GVL_Objects.List_of_Recipes[3].Compress.Initial_Speed :=  ConfigData.Rec3_Compress_Initial_Speed;
GVL_Objects.List_of_Recipes[3].Compress.Initial_Distance := ConfigData.Rec3_Compress_Initial_Distance;
GVL_Objects.List_of_Recipes[3].Compress.Shield_Dwell := ConfigData.Rec3_Compress_Shield_Dwell;
GVL_Objects.List_of_Recipes[3].Compress.Relax_Distance := ConfigData.Rec3_Compress_Relax_Distance;
GVL_Objects.List_of_Recipes[3].Compress.Retract_Speed := ConfigData.Rec3_Compress_Retract_Speed;

GVL_Objects.List_of_Recipes[3].Pusher.Initial_Speed := ConfigData.Rec3_Pusher_Initial_Speed;
GVL_Objects.List_of_Recipes[3].Pusher.Initial_Distance := ConfigData.Rec3_Pusher_Initial_Distance;
GVL_Objects.List_of_Recipes[3].Pusher.Eject_Speed := ConfigData.Rec3_Pusher_Eject_Speed;
GVL_Objects.List_of_Recipes[3].Pusher.Eject_Distance := ConfigData.Rec3_Pusher_Eject_Distance;
GVL_Objects.List_of_Recipes[3].Pusher.Retract_Speed := ConfigData.Rec3_Pusher_Retract_Speed;

GVL_Objects.List_of_Recipes[3].Pusher.tamp_final_distance := ConfigData.Rec3_Pusher_tamp_final_distance;
GVL_Objects.List_of_Recipes[3].Pusher.tamp_final_speed := ConfigData.Rec3_Pusher_tamp_final_speed;
GVL_Objects.List_of_Recipes[3].Pusher.tamp_initial_distance := ConfigData.Rec3_Pusher_tamp_initial_distance;
GVL_Objects.List_of_Recipes[3].Pusher.tamp_initial_speed := ConfigData.Rec3_Pusher_tamp_initial_speed;

GVL_Objects.List_of_Recipes[3].Other.Compress_Home_Offset := ConfigData.Other3_Compress_Home_Offset;
GVL_Objects.List_of_Recipes[3].Other.Pusher_Home_Offset := ConfigData.Other3_Pusher_Home_Offset;
GVL_Objects.List_of_Recipes[3].Other.Shield_Home_Offset := ConfigData.Other3_Shield_Home_Offset;
GVL_Objects.List_of_Recipes[3].Other.Axis_Acceleration := ConfigData.Other3_Axis_Acceleration;
GVL_Objects.List_of_Recipes[3].Other.Axis_Deceleration := ConfigData.Other3_Axis_Deceleration;
GVL_Objects.List_of_Recipes[3].Other.Axis_Jerk := ConfigData.Other3_Axis_Jerk;
GVL_Objects.List_of_Recipes[3].Memory_Free := LREAL_TO_BOOL(ConfigData.Other3_Memory_Free);

GVL_Objects.List_of_Recipes[3].Clamp.Release_Instance := ConfigData.Clamp3_Release_Instance;

Rec4_Name_1:=ConfigData.Rec4_Name_1;								
Rec4_Name_2:=ConfigData.Rec4_Name_2;								
Rec4_Name_3:=ConfigData.Rec4_Name_3;								
Rec4_Name_4:=ConfigData.Rec4_Name_4;								
Rec4_Name_5:=ConfigData.Rec4_Name_5;
List_of_Recipes[4].Name := Recipe_mem_4;

GVL_Objects.List_of_Recipes[4].Shield.Retract_Speed := ConfigData.Rec4_Shield_Retract_Speed;
GVL_Objects.List_of_Recipes[4].Shield.Initial_Speed := ConfigData.Rec4_Shield_Initial_Speed;
GVL_Objects.List_of_Recipes[4].Shield.Initial_Distance := ConfigData.Rec4_Shield_Initial_Distance;

GVL_Objects.List_of_Recipes[4].Compress.Initial_Speed :=  ConfigData.Rec4_Compress_Initial_Speed;
GVL_Objects.List_of_Recipes[4].Compress.Initial_Distance := ConfigData.Rec4_Compress_Initial_Distance;
GVL_Objects.List_of_Recipes[4].Compress.Shield_Dwell := ConfigData.Rec4_Compress_Shield_Dwell;
GVL_Objects.List_of_Recipes[4].Compress.Relax_Distance := ConfigData.Rec4_Compress_Relax_Distance;
GVL_Objects.List_of_Recipes[4].Compress.Retract_Speed := ConfigData.Rec4_Compress_Retract_Speed;

GVL_Objects.List_of_Recipes[4].Pusher.Initial_Speed := ConfigData.Rec4_Pusher_Initial_Speed;
GVL_Objects.List_of_Recipes[4].Pusher.Initial_Distance := ConfigData.Rec4_Pusher_Initial_Distance;
GVL_Objects.List_of_Recipes[4].Pusher.Eject_Speed := ConfigData.Rec4_Pusher_Eject_Speed;
GVL_Objects.List_of_Recipes[4].Pusher.Eject_Distance := ConfigData.Rec4_Pusher_Eject_Distance;
GVL_Objects.List_of_Recipes[4].Pusher.Retract_Speed := ConfigData.Rec4_Pusher_Retract_Speed;

GVL_Objects.List_of_Recipes[4].Pusher.tamp_final_distance := ConfigData.Rec4_Pusher_tamp_final_distance;
GVL_Objects.List_of_Recipes[4].Pusher.tamp_final_speed := ConfigData.Rec4_Pusher_tamp_final_speed;
GVL_Objects.List_of_Recipes[4].Pusher.tamp_initial_distance := ConfigData.Rec4_Pusher_tamp_initial_distance;
GVL_Objects.List_of_Recipes[4].Pusher.tamp_initial_speed := ConfigData.Rec4_Pusher_tamp_initial_speed;

GVL_Objects.List_of_Recipes[4].Other.Compress_Home_Offset := ConfigData.Other4_Compress_Home_Offset;
GVL_Objects.List_of_Recipes[4].Other.Pusher_Home_Offset := ConfigData.Other4_Pusher_Home_Offset;
GVL_Objects.List_of_Recipes[4].Other.Shield_Home_Offset := ConfigData.Other4_Shield_Home_Offset;
GVL_Objects.List_of_Recipes[4].Other.Axis_Acceleration := ConfigData.Other4_Axis_Acceleration;
GVL_Objects.List_of_Recipes[4].Other.Axis_Deceleration := ConfigData.Other4_Axis_Deceleration;
GVL_Objects.List_of_Recipes[4].Other.Axis_Jerk := ConfigData.Other4_Axis_Jerk;
GVL_Objects.List_of_Recipes[4].Memory_Free := LREAL_TO_BOOL(ConfigData.Other4_Memory_Free);

GVL_Objects.List_of_Recipes[4].Clamp.Release_Instance := ConfigData.Clamp4_Release_Instance;

Rec5_Name_1:=ConfigData.Rec5_Name_1;								
Rec5_Name_2:=ConfigData.Rec5_Name_2;								
Rec5_Name_3:=ConfigData.Rec5_Name_3;								
Rec5_Name_4:=ConfigData.Rec5_Name_4;								
Rec5_Name_5:=ConfigData.Rec5_Name_5;
List_of_Recipes[5].Name := Recipe_mem_5;

GVL_Objects.List_of_Recipes[5].Shield.Retract_Speed := ConfigData.Rec5_Shield_Retract_Speed;
GVL_Objects.List_of_Recipes[5].Shield.Initial_Speed := ConfigData.Rec5_Shield_Initial_Speed;
GVL_Objects.List_of_Recipes[5].Shield.Initial_Distance := ConfigData.Rec5_Shield_Initial_Distance;

GVL_Objects.List_of_Recipes[5].Compress.Initial_Speed :=  ConfigData.Rec5_Compress_Initial_Speed;
GVL_Objects.List_of_Recipes[5].Compress.Initial_Distance := ConfigData.Rec5_Compress_Initial_Distance;
GVL_Objects.List_of_Recipes[5].Compress.Shield_Dwell := ConfigData.Rec5_Compress_Shield_Dwell;
GVL_Objects.List_of_Recipes[5].Compress.Relax_Distance := ConfigData.Rec5_Compress_Relax_Distance;
GVL_Objects.List_of_Recipes[5].Compress.Retract_Speed := ConfigData.Rec5_Compress_Retract_Speed;

GVL_Objects.List_of_Recipes[5].Pusher.Initial_Speed := ConfigData.Rec5_Pusher_Initial_Speed;
GVL_Objects.List_of_Recipes[5].Pusher.Initial_Distance := ConfigData.Rec5_Pusher_Initial_Distance;
GVL_Objects.List_of_Recipes[5].Pusher.Eject_Speed := ConfigData.Rec5_Pusher_Eject_Speed;
GVL_Objects.List_of_Recipes[5].Pusher.Eject_Distance := ConfigData.Rec5_Pusher_Eject_Distance;
GVL_Objects.List_of_Recipes[5].Pusher.Retract_Speed := ConfigData.Rec5_Pusher_Retract_Speed;

GVL_Objects.List_of_Recipes[5].Pusher.tamp_final_distance := ConfigData.Rec5_Pusher_tamp_final_distance;
GVL_Objects.List_of_Recipes[5].Pusher.tamp_final_speed := ConfigData.Rec5_Pusher_tamp_final_speed;
GVL_Objects.List_of_Recipes[5].Pusher.tamp_initial_distance := ConfigData.Rec5_Pusher_tamp_initial_distance;
GVL_Objects.List_of_Recipes[5].Pusher.tamp_initial_speed := ConfigData.Rec5_Pusher_tamp_initial_speed;

GVL_Objects.List_of_Recipes[5].Other.Compress_Home_Offset := ConfigData.Other5_Compress_Home_Offset;
GVL_Objects.List_of_Recipes[5].Other.Pusher_Home_Offset := ConfigData.Other5_Pusher_Home_Offset;
GVL_Objects.List_of_Recipes[5].Other.Shield_Home_Offset := ConfigData.Other5_Shield_Home_Offset;
GVL_Objects.List_of_Recipes[5].Other.Axis_Acceleration := ConfigData.Other5_Axis_Acceleration;
GVL_Objects.List_of_Recipes[5].Other.Axis_Deceleration := ConfigData.Other5_Axis_Deceleration;
GVL_Objects.List_of_Recipes[5].Other.Axis_Jerk := ConfigData.Other5_Axis_Jerk;
GVL_Objects.List_of_Recipes[5].Memory_Free := LREAL_TO_BOOL(ConfigData.Other5_Memory_Free);

GVL_Objects.List_of_Recipes[5].Clamp.Release_Instance := ConfigData.Clamp5_Release_Instance;

Rec6_Name_1:=ConfigData.Rec6_Name_1;								
Rec6_Name_2:=ConfigData.Rec6_Name_2;								
Rec6_Name_3:=ConfigData.Rec6_Name_3;								
Rec6_Name_4:=ConfigData.Rec6_Name_4;								
Rec6_Name_5:=ConfigData.Rec6_Name_5;
List_of_Recipes[6].Name := Recipe_mem_6;

GVL_Objects.List_of_Recipes[6].Shield.Retract_Speed := ConfigData.Rec6_Shield_Retract_Speed;
GVL_Objects.List_of_Recipes[6].Shield.Initial_Speed := ConfigData.Rec6_Shield_Initial_Speed;
GVL_Objects.List_of_Recipes[6].Shield.Initial_Distance := ConfigData.Rec6_Shield_Initial_Distance;

GVL_Objects.List_of_Recipes[6].Compress.Initial_Speed :=  ConfigData.Rec6_Compress_Initial_Speed;
GVL_Objects.List_of_Recipes[6].Compress.Initial_Distance := ConfigData.Rec6_Compress_Initial_Distance;
GVL_Objects.List_of_Recipes[6].Compress.Shield_Dwell := ConfigData.Rec6_Compress_Shield_Dwell;
GVL_Objects.List_of_Recipes[6].Compress.Relax_Distance := ConfigData.Rec6_Compress_Relax_Distance;
GVL_Objects.List_of_Recipes[6].Compress.Retract_Speed := ConfigData.Rec6_Compress_Retract_Speed;

GVL_Objects.List_of_Recipes[6].Pusher.Initial_Speed := ConfigData.Rec6_Pusher_Initial_Speed;
GVL_Objects.List_of_Recipes[6].Pusher.Initial_Distance := ConfigData.Rec6_Pusher_Initial_Distance;
GVL_Objects.List_of_Recipes[6].Pusher.Eject_Speed := ConfigData.Rec6_Pusher_Eject_Speed;
GVL_Objects.List_of_Recipes[6].Pusher.Eject_Distance := ConfigData.Rec6_Pusher_Eject_Distance;
GVL_Objects.List_of_Recipes[6].Pusher.Retract_Speed := ConfigData.Rec6_Pusher_Retract_Speed;

GVL_Objects.List_of_Recipes[6].Pusher.tamp_final_distance := ConfigData.Rec6_Pusher_tamp_final_distance;
GVL_Objects.List_of_Recipes[6].Pusher.tamp_final_speed := ConfigData.Rec6_Pusher_tamp_final_speed;
GVL_Objects.List_of_Recipes[6].Pusher.tamp_initial_distance := ConfigData.Rec6_Pusher_tamp_initial_distance;
GVL_Objects.List_of_Recipes[6].Pusher.tamp_initial_speed := ConfigData.Rec6_Pusher_tamp_initial_speed;

GVL_Objects.List_of_Recipes[6].Other.Compress_Home_Offset := ConfigData.Other6_Compress_Home_Offset;
GVL_Objects.List_of_Recipes[6].Other.Pusher_Home_Offset := ConfigData.Other6_Pusher_Home_Offset;
GVL_Objects.List_of_Recipes[6].Other.Shield_Home_Offset := ConfigData.Other6_Shield_Home_Offset;
GVL_Objects.List_of_Recipes[6].Other.Axis_Acceleration := ConfigData.Other6_Axis_Acceleration;
GVL_Objects.List_of_Recipes[6].Other.Axis_Deceleration := ConfigData.Other6_Axis_Deceleration;
GVL_Objects.List_of_Recipes[6].Other.Axis_Jerk := ConfigData.Other6_Axis_Jerk;
GVL_Objects.List_of_Recipes[6].Memory_Free := LREAL_TO_BOOL(ConfigData.Other6_Memory_Free);

GVL_Objects.List_of_Recipes[6].Clamp.Release_Instance := ConfigData.Clamp6_Release_Instance;

Rec7_Name_1:=ConfigData.Rec7_Name_1;								
Rec7_Name_2:=ConfigData.Rec7_Name_2;								
Rec7_Name_3:=ConfigData.Rec7_Name_3;								
Rec7_Name_4:=ConfigData.Rec7_Name_4;								
Rec7_Name_5:=ConfigData.Rec7_Name_5;
List_of_Recipes[7].Name := Recipe_mem_7;

GVL_Objects.List_of_Recipes[7].Shield.Retract_Speed := ConfigData.Rec7_Shield_Retract_Speed;
GVL_Objects.List_of_Recipes[7].Shield.Initial_Speed := ConfigData.Rec7_Shield_Initial_Speed;
GVL_Objects.List_of_Recipes[7].Shield.Initial_Distance := ConfigData.Rec7_Shield_Initial_Distance;

GVL_Objects.List_of_Recipes[7].Compress.Initial_Speed :=  ConfigData.Rec7_Compress_Initial_Speed;
GVL_Objects.List_of_Recipes[7].Compress.Initial_Distance := ConfigData.Rec7_Compress_Initial_Distance;
GVL_Objects.List_of_Recipes[7].Compress.Shield_Dwell := ConfigData.Rec7_Compress_Shield_Dwell;
GVL_Objects.List_of_Recipes[7].Compress.Relax_Distance := ConfigData.Rec7_Compress_Relax_Distance;
GVL_Objects.List_of_Recipes[7].Compress.Retract_Speed := ConfigData.Rec7_Compress_Retract_Speed;

GVL_Objects.List_of_Recipes[7].Pusher.Initial_Speed := ConfigData.Rec7_Pusher_Initial_Speed;
GVL_Objects.List_of_Recipes[7].Pusher.Initial_Distance := ConfigData.Rec7_Pusher_Initial_Distance;
GVL_Objects.List_of_Recipes[7].Pusher.Eject_Speed := ConfigData.Rec7_Pusher_Eject_Speed;
GVL_Objects.List_of_Recipes[7].Pusher.Eject_Distance := ConfigData.Rec7_Pusher_Eject_Distance;
GVL_Objects.List_of_Recipes[7].Pusher.Retract_Speed := ConfigData.Rec7_Pusher_Retract_Speed;

GVL_Objects.List_of_Recipes[7].Pusher.tamp_final_distance := ConfigData.Rec7_Pusher_tamp_final_distance;
GVL_Objects.List_of_Recipes[7].Pusher.tamp_final_speed := ConfigData.Rec7_Pusher_tamp_final_speed;
GVL_Objects.List_of_Recipes[7].Pusher.tamp_initial_distance := ConfigData.Rec7_Pusher_tamp_initial_distance;
GVL_Objects.List_of_Recipes[7].Pusher.tamp_initial_speed := ConfigData.Rec7_Pusher_tamp_initial_speed;

GVL_Objects.List_of_Recipes[7].Other.Compress_Home_Offset := ConfigData.Other7_Compress_Home_Offset;
GVL_Objects.List_of_Recipes[7].Other.Pusher_Home_Offset := ConfigData.Other7_Pusher_Home_Offset;
GVL_Objects.List_of_Recipes[7].Other.Shield_Home_Offset := ConfigData.Other7_Shield_Home_Offset;
GVL_Objects.List_of_Recipes[7].Other.Axis_Acceleration := ConfigData.Other7_Axis_Acceleration;
GVL_Objects.List_of_Recipes[7].Other.Axis_Deceleration := ConfigData.Other7_Axis_Deceleration;
GVL_Objects.List_of_Recipes[7].Other.Axis_Jerk := ConfigData.Other7_Axis_Jerk;
GVL_Objects.List_of_Recipes[7].Memory_Free := LREAL_TO_BOOL(ConfigData.Other7_Memory_Free);

GVL_Objects.List_of_Recipes[7].Clamp.Release_Instance := ConfigData.Clamp7_Release_Instance;

Rec8_Name_1:=ConfigData.Rec8_Name_1;								
Rec8_Name_2:=ConfigData.Rec8_Name_2;								
Rec8_Name_3:=ConfigData.Rec8_Name_3;								
Rec8_Name_4:=ConfigData.Rec8_Name_4;								
Rec8_Name_5:=ConfigData.Rec8_Name_5;
List_of_Recipes[8].Name := Recipe_mem_8;

GVL_Objects.List_of_Recipes[8].Shield.Retract_Speed := ConfigData.Rec8_Shield_Retract_Speed;
GVL_Objects.List_of_Recipes[8].Shield.Initial_Speed := ConfigData.Rec8_Shield_Initial_Speed;
GVL_Objects.List_of_Recipes[8].Shield.Initial_Distance := ConfigData.Rec8_Shield_Initial_Distance;

GVL_Objects.List_of_Recipes[8].Compress.Initial_Speed :=  ConfigData.Rec8_Compress_Initial_Speed;
GVL_Objects.List_of_Recipes[8].Compress.Initial_Distance := ConfigData.Rec8_Compress_Initial_Distance;
GVL_Objects.List_of_Recipes[8].Compress.Shield_Dwell := ConfigData.Rec8_Compress_Shield_Dwell;
GVL_Objects.List_of_Recipes[8].Compress.Relax_Distance := ConfigData.Rec8_Compress_Relax_Distance;
GVL_Objects.List_of_Recipes[8].Compress.Retract_Speed := ConfigData.Rec8_Compress_Retract_Speed;

GVL_Objects.List_of_Recipes[8].Pusher.Initial_Speed := ConfigData.Rec8_Pusher_Initial_Speed;
GVL_Objects.List_of_Recipes[8].Pusher.Initial_Distance := ConfigData.Rec8_Pusher_Initial_Distance;
GVL_Objects.List_of_Recipes[8].Pusher.Eject_Speed := ConfigData.Rec8_Pusher_Eject_Speed;
GVL_Objects.List_of_Recipes[8].Pusher.Eject_Distance := ConfigData.Rec8_Pusher_Eject_Distance;
GVL_Objects.List_of_Recipes[8].Pusher.Retract_Speed := ConfigData.Rec8_Pusher_Retract_Speed;

GVL_Objects.List_of_Recipes[8].Pusher.tamp_final_distance := ConfigData.Rec8_Pusher_tamp_final_distance;
GVL_Objects.List_of_Recipes[8].Pusher.tamp_final_speed := ConfigData.Rec8_Pusher_tamp_final_speed;
GVL_Objects.List_of_Recipes[8].Pusher.tamp_initial_distance := ConfigData.Rec8_Pusher_tamp_initial_distance;
GVL_Objects.List_of_Recipes[8].Pusher.tamp_initial_speed := ConfigData.Rec8_Pusher_tamp_initial_speed;

GVL_Objects.List_of_Recipes[8].Other.Compress_Home_Offset := ConfigData.Other8_Compress_Home_Offset;
GVL_Objects.List_of_Recipes[8].Other.Pusher_Home_Offset := ConfigData.Other8_Pusher_Home_Offset;
GVL_Objects.List_of_Recipes[8].Other.Shield_Home_Offset := ConfigData.Other8_Shield_Home_Offset;
GVL_Objects.List_of_Recipes[8].Other.Axis_Acceleration := ConfigData.Other8_Axis_Acceleration;
GVL_Objects.List_of_Recipes[8].Other.Axis_Deceleration := ConfigData.Other8_Axis_Deceleration;
GVL_Objects.List_of_Recipes[8].Other.Axis_Jerk := ConfigData.Other8_Axis_Jerk;
GVL_Objects.List_of_Recipes[8].Memory_Free := LREAL_TO_BOOL(ConfigData.Other8_Memory_Free);

GVL_Objects.List_of_Recipes[8].Clamp.Release_Instance := ConfigData.Clamp8_Release_Instance;

Rec9_Name_1:=ConfigData.Rec9_Name_1;								
Rec9_Name_2:=ConfigData.Rec9_Name_2;								
Rec9_Name_3:=ConfigData.Rec9_Name_3;								
Rec9_Name_4:=ConfigData.Rec9_Name_4;								
Rec9_Name_5:=ConfigData.Rec9_Name_5;
List_of_Recipes[9].Name := Recipe_mem_9;

GVL_Objects.List_of_Recipes[9].Shield.Retract_Speed := ConfigData.Rec9_Shield_Retract_Speed;
GVL_Objects.List_of_Recipes[9].Shield.Initial_Speed := ConfigData.Rec9_Shield_Initial_Speed;
GVL_Objects.List_of_Recipes[9].Shield.Initial_Distance := ConfigData.Rec9_Shield_Initial_Distance;

GVL_Objects.List_of_Recipes[9].Compress.Initial_Speed :=  ConfigData.Rec9_Compress_Initial_Speed;
GVL_Objects.List_of_Recipes[9].Compress.Initial_Distance := ConfigData.Rec9_Compress_Initial_Distance;
GVL_Objects.List_of_Recipes[9].Compress.Shield_Dwell := ConfigData.Rec9_Compress_Shield_Dwell;
GVL_Objects.List_of_Recipes[9].Compress.Relax_Distance := ConfigData.Rec9_Compress_Relax_Distance;
GVL_Objects.List_of_Recipes[9].Compress.Retract_Speed := ConfigData.Rec9_Compress_Retract_Speed;

GVL_Objects.List_of_Recipes[9].Pusher.Initial_Speed := ConfigData.Rec9_Pusher_Initial_Speed;
GVL_Objects.List_of_Recipes[9].Pusher.Initial_Distance := ConfigData.Rec9_Pusher_Initial_Distance;
GVL_Objects.List_of_Recipes[9].Pusher.Eject_Speed := ConfigData.Rec9_Pusher_Eject_Speed;
GVL_Objects.List_of_Recipes[9].Pusher.Eject_Distance := ConfigData.Rec9_Pusher_Eject_Distance;
GVL_Objects.List_of_Recipes[9].Pusher.Retract_Speed := ConfigData.Rec9_Pusher_Retract_Speed;

GVL_Objects.List_of_Recipes[9].Pusher.tamp_final_distance := ConfigData.Rec9_Pusher_tamp_final_distance;
GVL_Objects.List_of_Recipes[9].Pusher.tamp_final_speed := ConfigData.Rec9_Pusher_tamp_final_speed;
GVL_Objects.List_of_Recipes[9].Pusher.tamp_initial_distance := ConfigData.Rec9_Pusher_tamp_initial_distance;
GVL_Objects.List_of_Recipes[9].Pusher.tamp_initial_speed := ConfigData.Rec9_Pusher_tamp_initial_speed;

GVL_Objects.List_of_Recipes[9].Other.Compress_Home_Offset := ConfigData.Other9_Compress_Home_Offset;
GVL_Objects.List_of_Recipes[9].Other.Pusher_Home_Offset := ConfigData.Other9_Pusher_Home_Offset;
GVL_Objects.List_of_Recipes[9].Other.Shield_Home_Offset := ConfigData.Other9_Shield_Home_Offset;
GVL_Objects.List_of_Recipes[9].Other.Axis_Acceleration := ConfigData.Other9_Axis_Acceleration;
GVL_Objects.List_of_Recipes[9].Other.Axis_Deceleration := ConfigData.Other9_Axis_Deceleration;
GVL_Objects.List_of_Recipes[9].Other.Axis_Jerk := ConfigData.Other9_Axis_Jerk;
GVL_Objects.List_of_Recipes[9].Memory_Free := LREAL_TO_BOOL(ConfigData.Other9_Memory_Free);

GVL_Objects.List_of_Recipes[9].Clamp.Release_Instance := ConfigData.Clamp9_Release_Instance;

Rec10_Name_1:=ConfigData.Rec10_Name_1;								
Rec10_Name_2:=ConfigData.Rec10_Name_2;								
Rec10_Name_3:=ConfigData.Rec10_Name_3;								
Rec10_Name_4:=ConfigData.Rec10_Name_4;								
Rec10_Name_5:=ConfigData.Rec10_Name_5;
List_of_Recipes[10].Name := Recipe_mem_10;

GVL_Objects.List_of_Recipes[10].Shield.Retract_Speed := ConfigData.Rec10_Shield_Retract_Speed;
GVL_Objects.List_of_Recipes[10].Shield.Initial_Speed := ConfigData.Rec10_Shield_Initial_Speed;
GVL_Objects.List_of_Recipes[10].Shield.Initial_Distance := ConfigData.Rec10_Shield_Initial_Distance;

GVL_Objects.List_of_Recipes[10].Compress.Initial_Speed :=  ConfigData.Rec10_Compress_Initial_Speed;
GVL_Objects.List_of_Recipes[10].Compress.Initial_Distance := ConfigData.Rec10_Compress_Initial_Distance;
GVL_Objects.List_of_Recipes[10].Compress.Shield_Dwell := ConfigData.Rec10_Compress_Shield_Dwell;
GVL_Objects.List_of_Recipes[10].Compress.Relax_Distance := ConfigData.Rec10_Compress_Relax_Distance;
GVL_Objects.List_of_Recipes[10].Compress.Retract_Speed := ConfigData.Rec10_Compress_Retract_Speed;

GVL_Objects.List_of_Recipes[10].Pusher.Initial_Speed := ConfigData.Rec10_Pusher_Initial_Speed;
GVL_Objects.List_of_Recipes[10].Pusher.Initial_Distance := ConfigData.Rec10_Pusher_Initial_Distance;
GVL_Objects.List_of_Recipes[10].Pusher.Eject_Speed := ConfigData.Rec10_Pusher_Eject_Speed;
GVL_Objects.List_of_Recipes[10].Pusher.Eject_Distance := ConfigData.Rec10_Pusher_Eject_Distance;
GVL_Objects.List_of_Recipes[10].Pusher.Retract_Speed := ConfigData.Rec10_Pusher_Retract_Speed;

GVL_Objects.List_of_Recipes[10].Pusher.tamp_final_distance := ConfigData.Rec10_Pusher_tamp_final_distance;
GVL_Objects.List_of_Recipes[10].Pusher.tamp_final_speed := ConfigData.Rec10_Pusher_tamp_final_speed;
GVL_Objects.List_of_Recipes[10].Pusher.tamp_initial_distance := ConfigData.Rec10_Pusher_tamp_initial_distance;
GVL_Objects.List_of_Recipes[10].Pusher.tamp_initial_speed := ConfigData.Rec10_Pusher_tamp_initial_speed;

GVL_Objects.List_of_Recipes[10].Other.Compress_Home_Offset := ConfigData.Other10_Compress_Home_Offset;
GVL_Objects.List_of_Recipes[10].Other.Pusher_Home_Offset := ConfigData.Other10_Pusher_Home_Offset;
GVL_Objects.List_of_Recipes[10].Other.Shield_Home_Offset := ConfigData.Other10_Shield_Home_Offset;
GVL_Objects.List_of_Recipes[10].Other.Axis_Acceleration := ConfigData.Other10_Axis_Acceleration;
GVL_Objects.List_of_Recipes[10].Other.Axis_Deceleration := ConfigData.Other10_Axis_Deceleration;
GVL_Objects.List_of_Recipes[10].Other.Axis_Jerk := ConfigData.Other10_Axis_Jerk;
GVL_Objects.List_of_Recipes[10].Memory_Free := LREAL_TO_BOOL(ConfigData.Other10_Memory_Free);

GVL_Objects.List_of_Recipes[10].Clamp.Release_Instance := ConfigData.Clamp10_Release_Instance;


//limits
GVL_Zenon.limits_save.max_limit_Compress := ConfigData.con_max_limit_Compress ; 					
GVL_Zenon.limits_save.max_limit_Shield := ConfigData.con_max_limit_Shield; 					
GVL_Zenon.limits_save.max_limit_Pusher := ConfigData.con_max_limit_Pusher;					
GVL_Zenon.limits_save.max_pusher_shield_diff := ConfigData.con_max_pusher_shield_diff;
END_METHOD

METHOD CopyConfigSettingsToGlobal : BOOL
VAR_INPUT
END_VAR
END_METHOD

METHOD CopyGlobalRecipiesToConfig : BOOL
VAR_INPUT
END_VAR
//ConfigData.Rec1_Name := GVL_Objects.List_of_Recipes[1].Name;

 
Recipe_mem_1:= List_of_Recipes[1].Name;

ConfigData.Rec1_Name_1:=Rec1_Name_1;								
ConfigData.Rec1_Name_2:=Rec1_Name_2;								
ConfigData.Rec1_Name_3:=Rec1_Name_3;								
ConfigData.Rec1_Name_4:=Rec1_Name_4;								
ConfigData.Rec1_Name_5:=Rec1_Name_5;	

ConfigData.Rec1_Shield_Retract_Speed := GVL_Objects.List_of_Recipes[1].Shield.Retract_Speed;
ConfigData.Rec1_Shield_Initial_Speed := GVL_Objects.List_of_Recipes[1].Shield.Initial_Speed;
ConfigData.Rec1_Shield_Initial_Distance := GVL_Objects.List_of_Recipes[1].Shield.Initial_distance;

ConfigData.Rec1_Compress_Initial_Speed := GVL_Objects.List_of_Recipes[1].Compress.Initial_Speed;
ConfigData.Rec1_Compress_Initial_Distance := GVL_Objects.List_of_Recipes[1].Compress.Initial_Distance;
ConfigData.Rec1_Compress_Shield_Dwell := GVL_Objects.List_of_Recipes[1].Compress.Shield_Dwell;
ConfigData.Rec1_Compress_Relax_Distance := GVL_Objects.List_of_Recipes[1].Compress.Relax_Distance;
ConfigData.Rec1_Compress_Retract_Speed := GVL_Objects.List_of_Recipes[1].Compress.Retract_Speed;


ConfigData.Rec1_Pusher_Initial_Speed := GVL_Objects.List_of_Recipes[1].Pusher.Initial_Speed;
ConfigData.Rec1_Pusher_Initial_Distance := GVL_Objects.List_of_Recipes[1].Pusher.Initial_Distance;
ConfigData.Rec1_Pusher_Eject_Speed := GVL_Objects.List_of_Recipes[1].Pusher.Eject_Speed;
ConfigData.Rec1_Pusher_Eject_Distance := GVL_Objects.List_of_Recipes[1].Pusher.Eject_Distance;
ConfigData.Rec1_Pusher_Retract_Speed := GVL_Objects.List_of_Recipes[1].Pusher.Retract_Speed;

ConfigData.Rec1_Pusher_tamp_initial_distance := GVL_Objects.List_of_Recipes[1].Pusher.tamp_initial_distance;
ConfigData.Rec1_Pusher_tamp_initial_speed := GVL_Objects.List_of_Recipes[1].Pusher.tamp_initial_speed;
ConfigData.Rec1_Pusher_tamp_final_distance := GVL_Objects.List_of_Recipes[1].Pusher.tamp_final_distance;
ConfigData.Rec1_Pusher_tamp_final_speed := GVL_Objects.List_of_Recipes[1].Pusher.tamp_final_speed;

ConfigData.Other1_Compress_Home_Offset := GVL_Objects.List_of_Recipes[1].Other.Compress_Home_Offset;
ConfigData.Other1_Pusher_Home_Offset := GVL_Objects.List_of_Recipes[1].Other.Pusher_Home_Offset;
ConfigData.Other1_Shield_Home_Offset := GVL_Objects.List_of_Recipes[1].Other.Shield_Home_Offset;
ConfigData.Other1_Axis_Acceleration := GVL_Objects.List_of_Recipes[1].Other.Axis_Acceleration;
ConfigData.Other1_Axis_Deceleration :=GVL_Objects.List_of_Recipes[1].Other.Axis_Deceleration;
ConfigData.Other1_Axis_Jerk := GVL_Objects.List_of_Recipes[1].Other.Axis_Jerk;
ConfigData.Other1_Memory_Free := BOOL_TO_LREAL(GVL_Objects.List_of_Recipes[1].Memory_Free);

ConfigData.Clamp1_Release_Instance := GVL_Objects.List_of_Recipes[1].Clamp.Release_Instance;

Recipe_mem_2:= List_of_Recipes[2].Name;
ConfigData.Rec2_Name_1:=Rec2_Name_1;								
ConfigData.Rec2_Name_2:=Rec2_Name_2;								
ConfigData.Rec2_Name_3:=Rec2_Name_3;								
ConfigData.Rec2_Name_4:=Rec2_Name_4;								
ConfigData.Rec2_Name_5:=Rec2_Name_5;

ConfigData.Rec2_Shield_Retract_Speed := GVL_Objects.List_of_Recipes[2].Shield.Retract_Speed;
ConfigData.Rec2_Shield_Initial_Speed := GVL_Objects.List_of_Recipes[2].Shield.Initial_Speed;
ConfigData.Rec2_Shield_Initial_Distance := GVL_Objects.List_of_Recipes[2].Shield.Initial_distance;

ConfigData.Rec2_Compress_Initial_Speed := GVL_Objects.List_of_Recipes[2].Compress.Initial_Speed;
ConfigData.Rec2_Compress_Initial_Distance := GVL_Objects.List_of_Recipes[2].Compress.Initial_Distance;
ConfigData.Rec2_Compress_Shield_Dwell := GVL_Objects.List_of_Recipes[2].Compress.Shield_Dwell;
ConfigData.Rec2_Compress_Relax_Distance := GVL_Objects.List_of_Recipes[2].Compress.Relax_Distance;
ConfigData.Rec2_Compress_Retract_Speed := GVL_Objects.List_of_Recipes[2].Compress.Retract_Speed;

ConfigData.Rec2_Pusher_Initial_Speed := GVL_Objects.List_of_Recipes[2].Pusher.Initial_Speed;
ConfigData.Rec2_Pusher_Initial_Distance := GVL_Objects.List_of_Recipes[2].Pusher.Initial_Distance;
ConfigData.Rec2_Pusher_Eject_Speed := GVL_Objects.List_of_Recipes[2].Pusher.Eject_Speed;
ConfigData.Rec2_Pusher_Eject_Distance := GVL_Objects.List_of_Recipes[2].Pusher.Eject_Distance;
ConfigData.Rec2_Pusher_Retract_Speed := GVL_Objects.List_of_Recipes[2].Pusher.Retract_Speed;

ConfigData.Rec2_Pusher_tamp_initial_distance := GVL_Objects.List_of_Recipes[2].Pusher.tamp_initial_distance;
ConfigData.Rec2_Pusher_tamp_initial_speed := GVL_Objects.List_of_Recipes[2].Pusher.tamp_initial_speed;
ConfigData.Rec2_Pusher_tamp_final_distance := GVL_Objects.List_of_Recipes[2].Pusher.tamp_final_distance;
ConfigData.Rec2_Pusher_tamp_final_speed := GVL_Objects.List_of_Recipes[2].Pusher.tamp_final_speed;

ConfigData.Other2_Compress_Home_Offset := GVL_Objects.List_of_Recipes[2].Other.Compress_Home_Offset;
ConfigData.Other2_Pusher_Home_Offset := GVL_Objects.List_of_Recipes[2].Other.Pusher_Home_Offset;
ConfigData.Other2_Shield_Home_Offset := GVL_Objects.List_of_Recipes[2].Other.Shield_Home_Offset;
ConfigData.Other2_Axis_Acceleration := GVL_Objects.List_of_Recipes[2].Other.Axis_Acceleration;
ConfigData.Other2_Axis_Deceleration :=GVL_Objects.List_of_Recipes[2].Other.Axis_Deceleration;
ConfigData.Other2_Axis_Jerk := GVL_Objects.List_of_Recipes[2].Other.Axis_Jerk;
ConfigData.Other2_Memory_Free := BOOL_TO_LREAL(GVL_Objects.List_of_Recipes[2].Memory_Free);

ConfigData.Clamp2_Release_Instance := GVL_Objects.List_of_Recipes[2].Clamp.Release_Instance;

Recipe_mem_3:= List_of_Recipes[3].Name;
ConfigData.Rec3_Name_1:=Rec3_Name_1;								
ConfigData.Rec3_Name_2:=Rec3_Name_2;								
ConfigData.Rec3_Name_3:=Rec3_Name_3;								
ConfigData.Rec3_Name_4:=Rec3_Name_4;								
ConfigData.Rec3_Name_5:=Rec3_Name_5;

ConfigData.Rec3_Shield_Retract_Speed := GVL_Objects.List_of_Recipes[3].Shield.Retract_Speed;
ConfigData.Rec3_Shield_Initial_Speed := GVL_Objects.List_of_Recipes[3].Shield.Initial_Speed;
ConfigData.Rec3_Shield_Initial_Distance := GVL_Objects.List_of_Recipes[3].Shield.Initial_distance;

ConfigData.Rec3_Compress_Initial_Speed := GVL_Objects.List_of_Recipes[3].Compress.Initial_Speed;
ConfigData.Rec3_Compress_Initial_Distance := GVL_Objects.List_of_Recipes[3].Compress.Initial_Distance;
ConfigData.Rec3_Compress_Shield_Dwell := GVL_Objects.List_of_Recipes[3].Compress.Shield_Dwell;
ConfigData.Rec3_Compress_Relax_Distance := GVL_Objects.List_of_Recipes[3].Compress.Relax_Distance;
ConfigData.Rec3_Compress_Retract_Speed := GVL_Objects.List_of_Recipes[3].Compress.Retract_Speed;

ConfigData.Rec3_Pusher_Initial_Speed := GVL_Objects.List_of_Recipes[3].Pusher.Initial_Speed;
ConfigData.Rec3_Pusher_Initial_Distance := GVL_Objects.List_of_Recipes[3].Pusher.Initial_Distance;
ConfigData.Rec3_Pusher_Eject_Speed := GVL_Objects.List_of_Recipes[3].Pusher.Eject_Speed;
ConfigData.Rec3_Pusher_Eject_Distance := GVL_Objects.List_of_Recipes[3].Pusher.Eject_Distance;
ConfigData.Rec3_Pusher_Retract_Speed := GVL_Objects.List_of_Recipes[3].Pusher.Retract_Speed;

ConfigData.Rec3_Pusher_tamp_initial_distance := GVL_Objects.List_of_Recipes[3].Pusher.tamp_initial_distance;
ConfigData.Rec3_Pusher_tamp_initial_speed := GVL_Objects.List_of_Recipes[3].Pusher.tamp_initial_speed;
ConfigData.Rec3_Pusher_tamp_final_distance := GVL_Objects.List_of_Recipes[3].Pusher.tamp_final_distance;
ConfigData.Rec3_Pusher_tamp_final_speed := GVL_Objects.List_of_Recipes[3].Pusher.tamp_final_speed;

ConfigData.Other3_Compress_Home_Offset := GVL_Objects.List_of_Recipes[3].Other.Compress_Home_Offset;
ConfigData.Other3_Pusher_Home_Offset := GVL_Objects.List_of_Recipes[3].Other.Pusher_Home_Offset;
ConfigData.Other3_Shield_Home_Offset := GVL_Objects.List_of_Recipes[3].Other.Shield_Home_Offset;
ConfigData.Other3_Axis_Acceleration := GVL_Objects.List_of_Recipes[3].Other.Axis_Acceleration;
ConfigData.Other3_Axis_Deceleration :=GVL_Objects.List_of_Recipes[3].Other.Axis_Deceleration;
ConfigData.Other3_Axis_Jerk := GVL_Objects.List_of_Recipes[3].Other.Axis_Jerk;
ConfigData.Other3_Memory_Free := BOOL_TO_LREAL(GVL_Objects.List_of_Recipes[3].Memory_Free);

ConfigData.Clamp3_Release_Instance := GVL_Objects.List_of_Recipes[3].Clamp.Release_Instance;

Recipe_mem_4:= List_of_Recipes[4].Name;
ConfigData.Rec4_Name_1:=Rec4_Name_1;								
ConfigData.Rec4_Name_2:=Rec4_Name_2;								
ConfigData.Rec4_Name_3:=Rec4_Name_3;								
ConfigData.Rec4_Name_4:=Rec4_Name_4;								
ConfigData.Rec4_Name_5:=Rec4_Name_5;

ConfigData.Rec4_Shield_Retract_Speed := GVL_Objects.List_of_Recipes[4].Shield.Retract_Speed;
ConfigData.Rec4_Shield_Initial_Speed := GVL_Objects.List_of_Recipes[4].Shield.Initial_Speed;
ConfigData.Rec4_Shield_Initial_Distance := GVL_Objects.List_of_Recipes[4].Shield.Initial_distance;

ConfigData.Rec4_Compress_Initial_Speed := GVL_Objects.List_of_Recipes[4].Compress.Initial_Speed;
ConfigData.Rec4_Compress_Initial_Distance := GVL_Objects.List_of_Recipes[4].Compress.Initial_Distance;
ConfigData.Rec4_Compress_Shield_Dwell := GVL_Objects.List_of_Recipes[4].Compress.Shield_Dwell;
ConfigData.Rec4_Compress_Relax_Distance := GVL_Objects.List_of_Recipes[4].Compress.Relax_Distance;
ConfigData.Rec4_Compress_Retract_Speed := GVL_Objects.List_of_Recipes[4].Compress.Retract_Speed;

ConfigData.Rec4_Pusher_Initial_Speed := GVL_Objects.List_of_Recipes[4].Pusher.Initial_Speed;
ConfigData.Rec4_Pusher_Initial_Distance := GVL_Objects.List_of_Recipes[4].Pusher.Initial_Distance;
ConfigData.Rec4_Pusher_Eject_Speed := GVL_Objects.List_of_Recipes[4].Pusher.Eject_Speed;
ConfigData.Rec4_Pusher_Eject_Distance := GVL_Objects.List_of_Recipes[4].Pusher.Eject_Distance;
ConfigData.Rec4_Pusher_Retract_Speed := GVL_Objects.List_of_Recipes[4].Pusher.Retract_Speed;

ConfigData.Rec4_Pusher_tamp_initial_distance := GVL_Objects.List_of_Recipes[4].Pusher.tamp_initial_distance;
ConfigData.Rec4_Pusher_tamp_initial_speed := GVL_Objects.List_of_Recipes[4].Pusher.tamp_initial_speed;
ConfigData.Rec4_Pusher_tamp_final_distance := GVL_Objects.List_of_Recipes[4].Pusher.tamp_final_distance;
ConfigData.Rec4_Pusher_tamp_final_speed := GVL_Objects.List_of_Recipes[4].Pusher.tamp_final_speed;

ConfigData.Other4_Compress_Home_Offset := GVL_Objects.List_of_Recipes[4].Other.Compress_Home_Offset;
ConfigData.Other4_Pusher_Home_Offset := GVL_Objects.List_of_Recipes[4].Other.Pusher_Home_Offset;
ConfigData.Other4_Shield_Home_Offset := GVL_Objects.List_of_Recipes[4].Other.Shield_Home_Offset;
ConfigData.Other4_Axis_Acceleration := GVL_Objects.List_of_Recipes[4].Other.Axis_Acceleration;
ConfigData.Other4_Axis_Deceleration :=GVL_Objects.List_of_Recipes[4].Other.Axis_Deceleration;
ConfigData.Other4_Axis_Jerk := GVL_Objects.List_of_Recipes[4].Other.Axis_Jerk;
ConfigData.Other4_Memory_Free := BOOL_TO_LREAL(GVL_Objects.List_of_Recipes[4].Memory_Free);

ConfigData.Clamp4_Release_Instance := GVL_Objects.List_of_Recipes[4].Clamp.Release_Instance;

Recipe_mem_5:= List_of_Recipes[5].Name;
ConfigData.Rec5_Name_1:=Rec5_Name_1;								
ConfigData.Rec5_Name_2:=Rec5_Name_2;								
ConfigData.Rec5_Name_3:=Rec5_Name_3;								
ConfigData.Rec5_Name_4:=Rec5_Name_4;								
ConfigData.Rec5_Name_5:=Rec5_Name_5;

ConfigData.Rec5_Shield_Retract_Speed := GVL_Objects.List_of_Recipes[5].Shield.Retract_Speed;
ConfigData.Rec5_Shield_Initial_Speed := GVL_Objects.List_of_Recipes[5].Shield.Initial_Speed;
ConfigData.Rec5_Shield_Initial_Distance := GVL_Objects.List_of_Recipes[5].Shield.Initial_distance;

ConfigData.Rec5_Compress_Initial_Speed := GVL_Objects.List_of_Recipes[5].Compress.Initial_Speed;
ConfigData.Rec5_Compress_Initial_Distance := GVL_Objects.List_of_Recipes[5].Compress.Initial_Distance;
ConfigData.Rec5_Compress_Shield_Dwell := GVL_Objects.List_of_Recipes[5].Compress.Shield_Dwell;
ConfigData.Rec5_Compress_Relax_Distance := GVL_Objects.List_of_Recipes[5].Compress.Relax_Distance;
ConfigData.Rec5_Compress_Retract_Speed := GVL_Objects.List_of_Recipes[5].Compress.Retract_Speed;

ConfigData.Rec5_Pusher_Initial_Speed := GVL_Objects.List_of_Recipes[5].Pusher.Initial_Speed;
ConfigData.Rec5_Pusher_Initial_Distance := GVL_Objects.List_of_Recipes[5].Pusher.Initial_Distance;
ConfigData.Rec5_Pusher_Eject_Speed := GVL_Objects.List_of_Recipes[5].Pusher.Eject_Speed;
ConfigData.Rec5_Pusher_Eject_Distance := GVL_Objects.List_of_Recipes[5].Pusher.Eject_Distance;
ConfigData.Rec5_Pusher_Retract_Speed := GVL_Objects.List_of_Recipes[5].Pusher.Retract_Speed;

ConfigData.Rec5_Pusher_tamp_initial_distance := GVL_Objects.List_of_Recipes[5].Pusher.tamp_initial_distance;
ConfigData.Rec5_Pusher_tamp_initial_speed := GVL_Objects.List_of_Recipes[5].Pusher.tamp_initial_speed;
ConfigData.Rec5_Pusher_tamp_final_distance := GVL_Objects.List_of_Recipes[5].Pusher.tamp_final_distance;
ConfigData.Rec5_Pusher_tamp_final_speed := GVL_Objects.List_of_Recipes[5].Pusher.tamp_final_speed;

ConfigData.Other5_Compress_Home_Offset := GVL_Objects.List_of_Recipes[5].Other.Compress_Home_Offset;
ConfigData.Other5_Pusher_Home_Offset := GVL_Objects.List_of_Recipes[5].Other.Pusher_Home_Offset;
ConfigData.Other5_Shield_Home_Offset := GVL_Objects.List_of_Recipes[5].Other.Shield_Home_Offset;
ConfigData.Other5_Axis_Acceleration := GVL_Objects.List_of_Recipes[5].Other.Axis_Acceleration;
ConfigData.Other5_Axis_Deceleration :=GVL_Objects.List_of_Recipes[5].Other.Axis_Deceleration;
ConfigData.Other5_Axis_Jerk := GVL_Objects.List_of_Recipes[5].Other.Axis_Jerk;
ConfigData.Other5_Memory_Free := BOOL_TO_LREAL(GVL_Objects.List_of_Recipes[5].Memory_Free);

ConfigData.Clamp5_Release_Instance := GVL_Objects.List_of_Recipes[5].Clamp.Release_Instance;

Recipe_mem_6:= List_of_Recipes[6].Name;
ConfigData.Rec6_Name_1:=Rec6_Name_1;								
ConfigData.Rec6_Name_2:=Rec6_Name_2;								
ConfigData.Rec6_Name_3:=Rec6_Name_3;								
ConfigData.Rec6_Name_4:=Rec6_Name_4;								
ConfigData.Rec6_Name_5:=Rec6_Name_5;

ConfigData.Rec6_Shield_Retract_Speed := GVL_Objects.List_of_Recipes[6].Shield.Retract_Speed;
ConfigData.Rec6_Shield_Initial_Speed := GVL_Objects.List_of_Recipes[6].Shield.Initial_Speed;
ConfigData.Rec6_Shield_Initial_Distance := GVL_Objects.List_of_Recipes[6].Shield.Initial_distance;

ConfigData.Rec6_Compress_Initial_Speed := GVL_Objects.List_of_Recipes[6].Compress.Initial_Speed;
ConfigData.Rec6_Compress_Initial_Distance := GVL_Objects.List_of_Recipes[6].Compress.Initial_Distance;
ConfigData.Rec6_Compress_Shield_Dwell := GVL_Objects.List_of_Recipes[6].Compress.Shield_Dwell;
ConfigData.Rec6_Compress_Relax_Distance := GVL_Objects.List_of_Recipes[6].Compress.Relax_Distance;
ConfigData.Rec6_Compress_Retract_Speed := GVL_Objects.List_of_Recipes[6].Compress.Retract_Speed;

ConfigData.Rec6_Pusher_Initial_Speed := GVL_Objects.List_of_Recipes[6].Pusher.Initial_Speed;
ConfigData.Rec6_Pusher_Initial_Distance := GVL_Objects.List_of_Recipes[6].Pusher.Initial_Distance;
ConfigData.Rec6_Pusher_Eject_Speed := GVL_Objects.List_of_Recipes[6].Pusher.Eject_Speed;
ConfigData.Rec6_Pusher_Eject_Distance := GVL_Objects.List_of_Recipes[6].Pusher.Eject_Distance;
ConfigData.Rec6_Pusher_Retract_Speed := GVL_Objects.List_of_Recipes[6].Pusher.Retract_Speed;

ConfigData.Rec6_Pusher_tamp_initial_distance := GVL_Objects.List_of_Recipes[6].Pusher.tamp_initial_distance;
ConfigData.Rec6_Pusher_tamp_initial_speed := GVL_Objects.List_of_Recipes[6].Pusher.tamp_initial_speed;
ConfigData.Rec6_Pusher_tamp_final_distance := GVL_Objects.List_of_Recipes[6].Pusher.tamp_final_distance;
ConfigData.Rec6_Pusher_tamp_final_speed := GVL_Objects.List_of_Recipes[6].Pusher.tamp_final_speed;

ConfigData.Other6_Compress_Home_Offset := GVL_Objects.List_of_Recipes[6].Other.Compress_Home_Offset;
ConfigData.Other6_Pusher_Home_Offset := GVL_Objects.List_of_Recipes[6].Other.Pusher_Home_Offset;
ConfigData.Other6_Shield_Home_Offset := GVL_Objects.List_of_Recipes[6].Other.Shield_Home_Offset;
ConfigData.Other6_Axis_Acceleration := GVL_Objects.List_of_Recipes[6].Other.Axis_Acceleration;
ConfigData.Other6_Axis_Deceleration :=GVL_Objects.List_of_Recipes[6].Other.Axis_Deceleration;
ConfigData.Other6_Axis_Jerk := GVL_Objects.List_of_Recipes[6].Other.Axis_Jerk;
ConfigData.Other6_Memory_Free := BOOL_TO_LREAL(GVL_Objects.List_of_Recipes[6].Memory_Free);

ConfigData.Clamp6_Release_Instance := GVL_Objects.List_of_Recipes[6].Clamp.Release_Instance;

Recipe_mem_7:= List_of_Recipes[7].Name;
ConfigData.Rec7_Name_1:=Rec7_Name_1;								
ConfigData.Rec7_Name_2:=Rec7_Name_2;								
ConfigData.Rec7_Name_3:=Rec7_Name_3;								
ConfigData.Rec7_Name_4:=Rec7_Name_4;								
ConfigData.Rec7_Name_5:=Rec7_Name_5;

ConfigData.Rec7_Shield_Retract_Speed := GVL_Objects.List_of_Recipes[7].Shield.Retract_Speed;
ConfigData.Rec7_Shield_Initial_Speed := GVL_Objects.List_of_Recipes[7].Shield.Initial_Speed;
ConfigData.Rec7_Shield_Initial_Distance := GVL_Objects.List_of_Recipes[7].Shield.Initial_distance;

ConfigData.Rec7_Compress_Initial_Speed := GVL_Objects.List_of_Recipes[7].Compress.Initial_Speed;
ConfigData.Rec7_Compress_Initial_Distance := GVL_Objects.List_of_Recipes[7].Compress.Initial_Distance;
ConfigData.Rec7_Compress_Shield_Dwell := GVL_Objects.List_of_Recipes[7].Compress.Shield_Dwell;
ConfigData.Rec7_Compress_Relax_Distance := GVL_Objects.List_of_Recipes[7].Compress.Relax_Distance;
ConfigData.Rec7_Compress_Retract_Speed := GVL_Objects.List_of_Recipes[7].Compress.Retract_Speed;

ConfigData.Rec7_Pusher_Initial_Speed := GVL_Objects.List_of_Recipes[7].Pusher.Initial_Speed;
ConfigData.Rec7_Pusher_Initial_Distance := GVL_Objects.List_of_Recipes[7].Pusher.Initial_Distance;
ConfigData.Rec7_Pusher_Eject_Speed := GVL_Objects.List_of_Recipes[7].Pusher.Eject_Speed;
ConfigData.Rec7_Pusher_Eject_Distance := GVL_Objects.List_of_Recipes[7].Pusher.Eject_Distance;
ConfigData.Rec7_Pusher_Retract_Speed := GVL_Objects.List_of_Recipes[7].Pusher.Retract_Speed;

ConfigData.Rec7_Pusher_tamp_initial_distance := GVL_Objects.List_of_Recipes[7].Pusher.tamp_initial_distance;
ConfigData.Rec7_Pusher_tamp_initial_speed := GVL_Objects.List_of_Recipes[7].Pusher.tamp_initial_speed;
ConfigData.Rec7_Pusher_tamp_final_distance := GVL_Objects.List_of_Recipes[7].Pusher.tamp_final_distance;
ConfigData.Rec7_Pusher_tamp_final_speed := GVL_Objects.List_of_Recipes[7].Pusher.tamp_final_speed;

ConfigData.Other7_Compress_Home_Offset := GVL_Objects.List_of_Recipes[7].Other.Compress_Home_Offset;
ConfigData.Other7_Pusher_Home_Offset := GVL_Objects.List_of_Recipes[7].Other.Pusher_Home_Offset;
ConfigData.Other7_Shield_Home_Offset := GVL_Objects.List_of_Recipes[7].Other.Shield_Home_Offset;
ConfigData.Other7_Axis_Acceleration := GVL_Objects.List_of_Recipes[7].Other.Axis_Acceleration;
ConfigData.Other7_Axis_Deceleration :=GVL_Objects.List_of_Recipes[7].Other.Axis_Deceleration;
ConfigData.Other7_Axis_Jerk := GVL_Objects.List_of_Recipes[7].Other.Axis_Jerk;
ConfigData.Other7_Memory_Free := BOOL_TO_LREAL(GVL_Objects.List_of_Recipes[7].Memory_Free);

ConfigData.Clamp7_Release_Instance := GVL_Objects.List_of_Recipes[7].Clamp.Release_Instance;

Recipe_mem_8:= List_of_Recipes[8].Name;
ConfigData.Rec8_Name_1:=Rec8_Name_1;								
ConfigData.Rec8_Name_2:=Rec8_Name_2;								
ConfigData.Rec8_Name_3:=Rec8_Name_3;								
ConfigData.Rec8_Name_4:=Rec8_Name_4;								
ConfigData.Rec8_Name_5:=Rec8_Name_5;

ConfigData.Rec8_Shield_Retract_Speed := GVL_Objects.List_of_Recipes[8].Shield.Retract_Speed;
ConfigData.Rec8_Shield_Initial_Speed := GVL_Objects.List_of_Recipes[8].Shield.Initial_Speed;
ConfigData.Rec8_Shield_Initial_Distance := GVL_Objects.List_of_Recipes[8].Shield.Initial_distance;

ConfigData.Rec8_Compress_Initial_Speed := GVL_Objects.List_of_Recipes[8].Compress.Initial_Speed;
ConfigData.Rec8_Compress_Initial_Distance := GVL_Objects.List_of_Recipes[8].Compress.Initial_Distance;
ConfigData.Rec8_Compress_Shield_Dwell := GVL_Objects.List_of_Recipes[8].Compress.Shield_Dwell;
ConfigData.Rec8_Compress_Relax_Distance := GVL_Objects.List_of_Recipes[8].Compress.Relax_Distance;
ConfigData.Rec8_Compress_Retract_Speed := GVL_Objects.List_of_Recipes[8].Compress.Retract_Speed;

ConfigData.Rec8_Pusher_Initial_Speed := GVL_Objects.List_of_Recipes[8].Pusher.Initial_Speed;
ConfigData.Rec8_Pusher_Initial_Distance := GVL_Objects.List_of_Recipes[8].Pusher.Initial_Distance;
ConfigData.Rec8_Pusher_Eject_Speed := GVL_Objects.List_of_Recipes[8].Pusher.Eject_Speed;
ConfigData.Rec8_Pusher_Eject_Distance := GVL_Objects.List_of_Recipes[8].Pusher.Eject_Distance;
ConfigData.Rec8_Pusher_Retract_Speed := GVL_Objects.List_of_Recipes[8].Pusher.Retract_Speed;

ConfigData.Rec8_Pusher_tamp_initial_distance := GVL_Objects.List_of_Recipes[8].Pusher.tamp_initial_distance;
ConfigData.Rec8_Pusher_tamp_initial_speed := GVL_Objects.List_of_Recipes[8].Pusher.tamp_initial_speed;
ConfigData.Rec8_Pusher_tamp_final_distance := GVL_Objects.List_of_Recipes[8].Pusher.tamp_final_distance;
ConfigData.Rec8_Pusher_tamp_final_speed := GVL_Objects.List_of_Recipes[8].Pusher.tamp_final_speed;

ConfigData.Other8_Compress_Home_Offset := GVL_Objects.List_of_Recipes[8].Other.Compress_Home_Offset;
ConfigData.Other8_Pusher_Home_Offset := GVL_Objects.List_of_Recipes[8].Other.Pusher_Home_Offset;
ConfigData.Other8_Shield_Home_Offset := GVL_Objects.List_of_Recipes[8].Other.Shield_Home_Offset;
ConfigData.Other8_Axis_Acceleration := GVL_Objects.List_of_Recipes[8].Other.Axis_Acceleration;
ConfigData.Other8_Axis_Deceleration :=GVL_Objects.List_of_Recipes[8].Other.Axis_Deceleration;
ConfigData.Other8_Axis_Jerk := GVL_Objects.List_of_Recipes[8].Other.Axis_Jerk;
ConfigData.Other8_Memory_Free := BOOL_TO_LREAL(GVL_Objects.List_of_Recipes[8].Memory_Free);

ConfigData.Clamp8_Release_Instance := GVL_Objects.List_of_Recipes[8].Clamp.Release_Instance;

Recipe_mem_9:= List_of_Recipes[9].Name;
ConfigData.Rec9_Name_1:=Rec9_Name_1;								
ConfigData.Rec9_Name_2:=Rec9_Name_2;								
ConfigData.Rec9_Name_3:=Rec9_Name_3;								
ConfigData.Rec9_Name_4:=Rec9_Name_4;								
ConfigData.Rec9_Name_5:=Rec9_Name_5;

ConfigData.Rec9_Shield_Retract_Speed := GVL_Objects.List_of_Recipes[9].Shield.Retract_Speed;
ConfigData.Rec9_Shield_Initial_Speed := GVL_Objects.List_of_Recipes[9].Shield.Initial_Speed;
ConfigData.Rec9_Shield_Initial_Distance := GVL_Objects.List_of_Recipes[9].Shield.Initial_distance;

ConfigData.Rec9_Compress_Initial_Speed := GVL_Objects.List_of_Recipes[9].Compress.Initial_Speed;
ConfigData.Rec9_Compress_Initial_Distance := GVL_Objects.List_of_Recipes[9].Compress.Initial_Distance;
ConfigData.Rec9_Compress_Shield_Dwell := GVL_Objects.List_of_Recipes[9].Compress.Shield_Dwell;
ConfigData.Rec9_Compress_Relax_Distance := GVL_Objects.List_of_Recipes[9].Compress.Relax_Distance;
ConfigData.Rec9_Compress_Retract_Speed := GVL_Objects.List_of_Recipes[9].Compress.Retract_Speed;

ConfigData.Rec9_Pusher_Initial_Speed := GVL_Objects.List_of_Recipes[9].Pusher.Initial_Speed;
ConfigData.Rec9_Pusher_Initial_Distance := GVL_Objects.List_of_Recipes[9].Pusher.Initial_Distance;
ConfigData.Rec9_Pusher_Eject_Speed := GVL_Objects.List_of_Recipes[9].Pusher.Eject_Speed;
ConfigData.Rec9_Pusher_Eject_Distance := GVL_Objects.List_of_Recipes[9].Pusher.Eject_Distance;
ConfigData.Rec9_Pusher_Retract_Speed := GVL_Objects.List_of_Recipes[9].Pusher.Retract_Speed;

ConfigData.Rec9_Pusher_tamp_initial_distance := GVL_Objects.List_of_Recipes[9].Pusher.tamp_initial_distance;
ConfigData.Rec9_Pusher_tamp_initial_speed := GVL_Objects.List_of_Recipes[9].Pusher.tamp_initial_speed;
ConfigData.Rec9_Pusher_tamp_final_distance := GVL_Objects.List_of_Recipes[9].Pusher.tamp_final_distance;
ConfigData.Rec9_Pusher_tamp_final_speed := GVL_Objects.List_of_Recipes[9].Pusher.tamp_final_speed;

ConfigData.Other9_Compress_Home_Offset := GVL_Objects.List_of_Recipes[9].Other.Compress_Home_Offset;
ConfigData.Other9_Pusher_Home_Offset := GVL_Objects.List_of_Recipes[9].Other.Pusher_Home_Offset;
ConfigData.Other9_Shield_Home_Offset := GVL_Objects.List_of_Recipes[9].Other.Shield_Home_Offset;
ConfigData.Other9_Axis_Acceleration := GVL_Objects.List_of_Recipes[9].Other.Axis_Acceleration;
ConfigData.Other9_Axis_Deceleration :=GVL_Objects.List_of_Recipes[9].Other.Axis_Deceleration;
ConfigData.Other9_Axis_Jerk := GVL_Objects.List_of_Recipes[9].Other.Axis_Jerk;
ConfigData.Other9_Memory_Free := BOOL_TO_LREAL(GVL_Objects.List_of_Recipes[9].Memory_Free);

ConfigData.Clamp9_Release_Instance := GVL_Objects.List_of_Recipes[9].Clamp.Release_Instance;

Recipe_mem_10:= List_of_Recipes[10].Name;
ConfigData.Rec10_Name_1:=Rec10_Name_1;								
ConfigData.Rec10_Name_2:=Rec10_Name_2;								
ConfigData.Rec10_Name_3:=Rec10_Name_3;								
ConfigData.Rec10_Name_4:=Rec10_Name_4;								
ConfigData.Rec10_Name_5:=Rec10_Name_5;

ConfigData.Rec10_Shield_Retract_Speed := GVL_Objects.List_of_Recipes[10].Shield.Retract_Speed;
ConfigData.Rec10_Shield_Initial_Speed := GVL_Objects.List_of_Recipes[10].Shield.Initial_Speed;
ConfigData.Rec10_Shield_Initial_Distance := GVL_Objects.List_of_Recipes[10].Shield.Initial_distance;

ConfigData.Rec10_Compress_Initial_Speed := GVL_Objects.List_of_Recipes[10].Compress.Initial_Speed;
ConfigData.Rec10_Compress_Initial_Distance := GVL_Objects.List_of_Recipes[10].Compress.Initial_Distance;
ConfigData.Rec10_Compress_Shield_Dwell := GVL_Objects.List_of_Recipes[10].Compress.Shield_Dwell;
ConfigData.Rec10_Compress_Relax_Distance := GVL_Objects.List_of_Recipes[10].Compress.Relax_Distance;
ConfigData.Rec10_Compress_Retract_Speed := GVL_Objects.List_of_Recipes[10].Compress.Retract_Speed;

ConfigData.Rec10_Pusher_Initial_Speed := GVL_Objects.List_of_Recipes[10].Pusher.Initial_Speed;
ConfigData.Rec10_Pusher_Initial_Distance := GVL_Objects.List_of_Recipes[10].Pusher.Initial_Distance;
ConfigData.Rec10_Pusher_Eject_Speed := GVL_Objects.List_of_Recipes[10].Pusher.Eject_Speed;
ConfigData.Rec10_Pusher_Eject_Distance := GVL_Objects.List_of_Recipes[10].Pusher.Eject_Distance;
ConfigData.Rec10_Pusher_Retract_Speed := GVL_Objects.List_of_Recipes[10].Pusher.Retract_Speed;

ConfigData.Rec10_Pusher_tamp_initial_distance := GVL_Objects.List_of_Recipes[10].Pusher.tamp_initial_distance;
ConfigData.Rec10_Pusher_tamp_initial_speed := GVL_Objects.List_of_Recipes[10].Pusher.tamp_initial_speed;
ConfigData.Rec10_Pusher_tamp_final_distance := GVL_Objects.List_of_Recipes[10].Pusher.tamp_final_distance;
ConfigData.Rec10_Pusher_tamp_final_speed := GVL_Objects.List_of_Recipes[10].Pusher.tamp_final_speed;

ConfigData.Other10_Compress_Home_Offset := GVL_Objects.List_of_Recipes[10].Other.Compress_Home_Offset;
ConfigData.Other10_Pusher_Home_Offset := GVL_Objects.List_of_Recipes[10].Other.Pusher_Home_Offset;
ConfigData.Other10_Shield_Home_Offset := GVL_Objects.List_of_Recipes[10].Other.Shield_Home_Offset;
ConfigData.Other10_Axis_Acceleration := GVL_Objects.List_of_Recipes[10].Other.Axis_Acceleration;
ConfigData.Other10_Axis_Deceleration :=GVL_Objects.List_of_Recipes[10].Other.Axis_Deceleration;
ConfigData.Other10_Axis_Jerk := GVL_Objects.List_of_Recipes[10].Other.Axis_Jerk;
ConfigData.Other10_Memory_Free := BOOL_TO_LREAL(GVL_Objects.List_of_Recipes[10].Memory_Free);

ConfigData.Clamp10_Release_Instance := GVL_Objects.List_of_Recipes[10].Clamp.Release_Instance;

//limits
ConfigData.con_max_limit_Compress := GVL_Zenon.limits_save.max_limit_Compress; 					
ConfigData.con_max_limit_Shield	:= GVL_Zenon.limits_save.max_limit_Shield; 					
ConfigData.con_max_limit_Pusher := GVL_Zenon.limits_save.max_limit_Pusher;					
ConfigData.con_max_pusher_shield_diff := GVL_Zenon.limits_save.max_pusher_shield_diff;
END_METHOD

METHOD CopyGlobalSettingsToConfig : BOOL
VAR_INPUT
END_VAR
END_METHOD

METHOD Initialised : BOOL
VAR_INPUT
END_VAR
Initialised := ConfigData.Initialised;
END_METHOD

METHOD METH : BOOL
VAR_INPUT
	str : STRING(80); 
	pos : INT; 
	pt : POINTER TO ARRAY[0..79] OF BYTE; 
	size : UINT; 
END_VAR
VAR
	ps : POINTER TO BYTE; 
	i: INT; 
	end: INT;
END_VAR


ps := ADR(str); 
end := MIN(pos + LEN(str) - 1,UINT_TO_INT(size)); 

FOR i := pos TO end DO 
	pt^[i] := ps^; 
	ps := ps + 1; 
END_FOR;
END_METHOD

END_FUNCTION_BLOCK

// ---- XML/FB_Retain.TcPOU
FUNCTION_BLOCK FB_Retain
VAR_INPUT
	bEnable							: BOOL;				(* Turns on the autosave function *)
	bRead							: BOOL;				(* forces a read of the data from disk *)
	bForceWrite						: BOOL;				(* Ignores wait timer and checksum to save the data now *)
	tDelayTime						: TIME;				(* minimum time between data writes to disk *)
	pData							: pvoid;			(* pointer to the data *)
	nDataSize						: DWORD;			(* size of the data *)
	xPath							: STRING;			(* XML path for the data file *)
	sfilename						: STRING;			(* Filename and path *)
END_VAR
VAR_OUTPUT
		bBusy						: BOOL;				(* Block is busy *)
	bReadDone						: BOOL;				(* Block has finshed reading *)
	bWriteDone						: BOOL;				(* Block has finished writing *)
	bError							: BOOL;				(* Block has finished with an error *)
	nErrorID						: DWORD;			(* Error code *)
	bReadOnce						: BOOL;				(* Initial read complete *)
END_VAR
VAR
		eState						: eXMLState;
	nCurrentCheckSum				: DWORD;
	nLastCheckSum					: DWORD;
	fbTrig							: R_TRIG;
	fbForceWriteTrig				: R_TRIG;
	fbWaitTimer						: TON;
	fbXmlSrvWrite					: FB_XmlSrvWrite;
	fbXmlSrvRead					: FB_XmlSrvRead;
	PreviousRecipe: WORD;
END_VAR

CASE eState OF
	eXMLState.eWait: (* Wait for the timer *)
		fbForceWriteTrig(CLK := bForceWrite);
		//fbWaitTimer(IN := bEnable AND bReadOnce, PT := tDelayTime);
		//IF fbWaitTimer.Q OR fbForceWriteTrig.Q THEN
		IF fbForceWriteTrig.Q THEN 	//JT added
			nCurrentCheckSum := F_CheckSum16(dwSrcAddr := pData, cbLen := nDataSize, wChkSum := 1);
			IF (nCurrentCheckSum <> nLastCheckSum) OR fbForceWriteTrig.Q THEN
				//SavingRecipeChanges	:= TRUE;
				nLastCheckSum := nCurrentCheckSum;
				eState := eResetWrite;
				bBusy := TRUE;
				bWriteDone := FALSE;
				bError := FALSE;
				nErrorID := 0;
			END_IF
			fbWaitTimer(IN := FALSE);
		END_IF
		fbTrig(CLK := bRead);
		IF fbTrig.Q THEN
			bBusy := TRUE;
			bReadDone := FALSE;
			bError := FALSE;
			bReadOnce := FALSE;
			eState := eResetRead;
			nErrorID := 0;
		END_IF
	(* -------------------------------- *)

	eResetWrite: (* Reset XML Server *)
		fbXmlSrvWrite(
			sNetId:= '',
			ePath:= PATH_GENERIC,
			nMode:= XMLSRV_ADDMISSING,
			pSymAddr:= pData,
			cbSymSize:= nDataSize,
			sFilePath:= sfilename,
			sXPath:= xPath,
			bExecute:= FALSE,
			tTimeout:= T#10S,
			bBusy=> ,
			bError=> ,
			nErrId=> nErrorID);
		eState := eWriteData;
	(* -------------------------------- *)

	eWriteData: (* Write XML Data *)
		fbXmlSrvWrite(
			sNetId:= '',
			ePath:= PATH_GENERIC,
			nMode:= XMLSRV_ADDMISSING,
			pSymAddr:= pData,
			cbSymSize:= nDataSize,
			sFilePath:= sfilename,
			sXPath:= xPath,
			bExecute:= TRUE,
			tTimeout:= T#10S,
			bBusy=> ,
			bError=> ,
			nErrId=> nErrorID);
		IF NOT fbXmlSrvWrite.bBusy AND NOT fbXmlSrvWrite.bError THEN
			eState := eXMLState.eWait;
			//SavingRecipeChanges := false;
			bBusy := FALSE;
			bError := FALSE;
			bWriteDone := TRUE;
		ELSIF NOT fbXmlSrvWrite.bBusy AND fbXmlSrvWrite.bError THEN
			eState := eXMLState.eWait;
			sSystemStateHi := F_DisplayText("Data Not Saved",0);
			bBusy := FALSE;
			bError := TRUE;
		END_IF
	(* -------------------------------- *)

	eResetRead: (* Reset Read *)
		fbXmlSrvRead(
			sNetId:= '',
			ePath:= PATH_GENERIC,
			nMode:= XMLSRV_ADDMISSING,
			pSymAddr:= pData,
			cbSymSize:= nDataSize,
			sFilePath:= sfilename,
			sXPath:= xPath,
			bExecute:= FALSE,
			tTimeout:= T#10S,
			bBusy=> ,
			bError=> ,
			nErrId=> nErrorID);
		eState := eReadData;
	(* -------------------------------- *)

	eReadData: (* Read *)
		fbXmlSrvRead(
			sNetId:= '',
			ePath:= PATH_GENERIC,
			nMode:= XMLSRV_ADDMISSING,
			pSymAddr:= pData,
			cbSymSize:= nDataSize,
			sFilePath:= sfilename,
			sXPath:= xPath,
			bExecute:= TRUE,
			tTimeout:= T#100S,
			bBusy=> ,
			bError=> ,
			nErrId=> nErrorID);
		IF NOT fbXmlSrvRead.bBusy AND NOT fbXmlSrvRead.bError THEN
			eState := eXMLState.eWait;
			bBusy := FALSE;
			bError := FALSE;
			bReadDone := TRUE;
			bReadOnce := TRUE;
		ELSIF NOT fbXmlSrvRead.bBusy AND fbXmlSrvRead.bError THEN
			eState := eXMLState.eWait;
			bBusy := FALSE;
			bError := TRUE;
			bReadOnce := TRUE;
		END_IF
	(* -------------------------------- *)
END_CASE

END_FUNCTION_BLOCK
